Universal Robots PolyScope program: pruebacambio.urp

Program pruebacambio (installation=instalacion_derecha_10_MAR_21 directory=/programs/nueva carpeta createdIn=5.6.0.90886 lastSavedIn=5.6.0.90886 robotSerialNumber=20195001785)
Calibrated DH parameters: a=[0.000107, -0.568984, -0.552934, -0.00001, -0.000063, 0]; d=[0.180718, -257.998067, 200.685024, 57.48776, 0.119923, 0.115353]; alpha=[1.571119, 0.000876, -0.002498, 1.571178, -1.570523, 0]; deltaTheta=[0, -0.378191, 0.631587, -0.253396, 0, 0]
Robot Program (runOnlyOnce=false)
  MoveJ speed 60 deg/s, acceleration 80 deg/s^2 (useActiveTCP=true) feature=Plane_5
    Waypoint Waypoint_1: TCP in base x=-555.565 y=-387.14 z=53.84 mm, rx=-1.9588 ry=2.3414 rz=-0.1116 rad; joints [24.639, -77.365, 117.778, -32.681, 115.442, 3.373] deg; TCP offset x=0.411 y=-218.298 z=37.994 mm, rx=1.558 ry=-0.1255 rz=0.1212 rad; feature pose in base x=-414.632 y=-364.771 z=-8.601 mm, rx=0.0051 ry=-3.1307 rz=0.001 rad
    y := .1
    rx := 1
    ry := .5
    o := p[0,y,0,rx,ry,0]
    Plane_5 := pose_trans(Plane_5, o)
  MoveJ speed 60 deg/s, acceleration 80 deg/s^2 (useActiveTCP=true) feature=Plane_5
    Waypoint Waypoint_1: TCP in base x=-555.565 y=-387.14 z=53.84 mm, rx=-1.9588 ry=2.3414 rz=-0.1116 rad; joints [24.639, -77.365, 117.778, -32.681, 115.442, 3.373] deg
    Waypoint Waypoint_3: TCP in base x=-658.118 y=-382.212 z=54.957 mm, rx=2.01 ry=-2.4028 rz=-0.0103 rad; joints [21.333, -73.182, 114.102, -41.079, 112.325, 0.146] deg; TCP offset x=0.411 y=-218.298 z=37.994 mm, rx=1.558 ry=-0.1255 rz=0.1212 rad; feature pose in base x=-414.632 y=-364.771 z=-8.601 mm, rx=0.0051 ry=-3.1307 rz=0.001 rad
